{attribute 'qualified_only'}
{attribute 'strict'}
TYPE E_NeedleClip :
(
	clip_A		:= 0,
	clip_B		:= 1,
	clip_C		:= 2,
	clip_D		:= 3,
);
END_TYPE

(* stored: Version 1.1.0.1, ProductVersion 3.1.4024.13
   DUT E_NeedleClip: Id {247ac1a5-661b-4af4-af5a-a66f45f2dd9b} *)
